Staubli VAL3: IfAbfrageController.pjx

Parameters version=s7.5.3 stackSize=5000 millimeterUnit=true
Program file=MoveJoint.pgx
Program file=MoveLine.pgx
Program file=start.pgx
Program file=stop.pgx
Program file=main.pgx
Data file=IfAbfrageController.dtx
